FUNCTION_BLOCK fbTest (* Basic Function Block Type *)
  (* Standard: 61499-2 *)
  (* Version 0.0, 10/1/2026, Schneider Electric, Template *)
  PACKAGE Main;
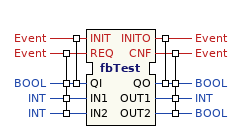
  EVENT_INPUT
    INIT WITH QI; (* Initialization Request *)
    REQ WITH QI, IN1, IN2; (* Normal Execution Request *)
  END_EVENT
  EVENT_OUTPUT
    INITO WITH QO; (* Initialization Confirm *)
    CNF WITH QO, OUT1, OUT2; (* Execution Confirmation *)
  END_EVENT
  VAR_INPUT
    QI : BOOL; (* Input event qualifier *)
    IN1 : INT;
    IN2 : INT;
  END_VAR
  VAR_OUTPUT
    QO : BOOL; (* Output event qualifier *)
    OUT1 : INT;
    OUT2 : BOOL;
  END_VAR
  VAR
    Counter : INT;
  END_VAR
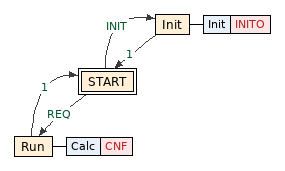
  EC_STATES
    START; (* Initial State *)
    Init : Init -> INITO; (* Initialization *)
    Run : Calc -> CNF; (* Normal execution *)
  END_STATES
  EC_TRANSITIONS
    START TO Init := INIT;
    Init TO START := 1;
    START TO Run := REQ;
    Run TO START := 1;
  END_TRANSITIONS
  ALGORITHM Init IN ST:
QO := QI;
Counter := 0;
  END_ALGORITHM
  ALGORITHM Calc IN ST:
Counter := Counter + 1;
OUT1 := IN1 + IN2;
OUT2 := OUT1 > 100;
  END_ALGORITHM
END_FUNCTION_BLOCK
